(* IEC 61131-3 sources: inproshop/TEAM_V2.0-demo_exported/2.Main, 6 files *)

(* ---- Main_Clock.st ---- *)
VAR_GLOBAL
	CPU_Clock:Str_Clock;
END_VAR

(* ---- Main_Communication.st ---- *)
VAR_GLOBAL
	From_OPXX AT %IW2000:Str_OP10_TO_OPXX;
	TO_OPXX AT %QW2000:Str_OPXX_TO_OP10;
	To_Slave:Str_ToSlave;

END_VAR

(* ---- Main_IO.st ---- *)
VAR_GLOBAL

END_VAR

VAR_GLOBAL

END_VAR

(* ---- Clock.st ---- *)
PROGRAM Clock
VAR
	data_clock_10ms:FB_Clock;
	data_clock_50ms:FB_Clock;
	data_clock_100ms:FB_Clock;
	data_clock_500ms:FB_Clock;
	data_clock_1s:FB_Clock;
END_VAR

//100MS脉冲
data_clock_10ms(iEnable:=TRUE,iClock:=1,o_Clock=>CPU_Clock.Clock_10ms);

//500MS脉冲
data_clock_50ms(iEnable:=TRUE,iClock:=5,o_Clock=>CPU_Clock.Clock_50ms);

//100MS脉冲
data_clock_100ms(iEnable:=TRUE,iClock:=10,o_Clock=>CPU_Clock.Clock_100ms);

//500MS脉冲
data_clock_500ms(iEnable:=TRUE,iClock:=50,o_Clock=>CPU_Clock.Clock_500ms);

//1S脉冲
data_clock_1s(iEnable:=TRUE,iClock:=100,o_Clock=>CPU_Clock.Clock_1s);

(* ---- PLC_PRG.st ---- *)
PROGRAM PLC_PRG
VAR
	Temp_pulse_on_R:R_TRIG;
	Temp_clock_10ms_R:R_TRIG;
	Temp_clock_50ms_R:R_TRIG;
	Temp_clock_100ms_R:R_TRIG;
	Temp_clock_500ms_R:R_TRIG;
	Temp_clock_1s_R:R_TRIG;

END_VAR
//RUN之后一个扫描周期ON
Temp_pulse_on_R(CLK:=TRUE,Q=>CPU_Clock.FirstRun);

//10ms脉冲上升沿
Temp_clock_10ms_R(CLK:=CPU_Clock.Clock_10ms,Q=>CPU_Clock.Clock_10ms_R);

//50ms脉冲上升沿
Temp_clock_50ms_R(CLK:=CPU_Clock.Clock_50ms,Q=>CPU_Clock.Clock_50ms_R);

//100ms脉冲上升沿
Temp_clock_100ms_R(CLK:=CPU_Clock.Clock_100ms,Q=>CPU_Clock.Clock_100ms_R);

//500ms脉冲上升沿
Temp_clock_500ms_R(CLK:=CPU_Clock.Clock_500ms,Q=>CPU_Clock.Clock_500ms_R);

//1s脉冲上升沿
Temp_clock_1s_R(CLK:=CPU_Clock.Clock_1s,Q=>CPU_Clock.Clock_1s_R);

//累计运行时间ms获取
GetSystemTime(udiTimeMs=>CPU_Clock.TimeMs );
//获取系统时间
GetSystemDate_sDt(stSystemDate=>CPU_Clock.DataToday);
//获取前31天时间
FC_SysTime(iNow:= CPU_Clock.DataToday, ioBefor:=CPU_Clock.DateOld );

//开班时间设定
CPU_Clock.DayStartTime:='8:30';
CPU_Clock.NightStartTime:='20:30';
//

OP10_Control();
OP11_Control();
OP20_Control();
OP30_Control();
OP70_Control();
OP80_Control();

(* ---- Test.st ---- *)
PROGRAM Test

VAR

	i:INT;
	PickPoint:INT;
END_VAR
